// TIA Portal V19 export
TYPE "PosFbk_ITF"
// stored: Access Published
   STRUCT
      Sts : Struct
         Error : Bool;
         ErrorNotSynched : Bool;
         PresetAck : Bool;
         EncIsAbsolute : Bool;
         Position : LReal;
      END_STRUCT;
      Ctrl : Struct
         Rst : Bool;
         PresetCmd : Bool;
         PresetPosition : LReal;
      END_STRUCT;
   END_STRUCT;
END_TYPE
